FUNCTION_BLOCK CON_LoadingStation
VAR_INPUT
	i_weighbridge 					: MOD_Loadingstation_I_stWeighbridge;
	i_tempIWantExtraBoxInTruck 		: BOOL;
	i_resetTime						: TIME := T#2S;//time necessary for the slowest part to reset
END_VAR
VAR_OUTPUT
	q_crane 						: MOD_Loadingstation_Q_stCrane;
END_VAR
VAR_IN_OUT
	iq_CommandState 				: INT;
END_VAR
VAR
	resetTimer						: TON;
	resetState 						: INT;
END_VAR

//check if there is a truck before running. Also check for weightlimit
IF NOT i_weighbridge.TruckOnScale THEN
	q_crane.AllowedToOperate 	:= FALSE;
	iq_CommandState 			:= Command.Abort; //Abort no truck
	
ELSIF i_weighbridge.TruckOnScale AND NOT i_weighbridge.WeightLimitReached THEN
	q_crane.AllowedToOperate 	:= TRUE;//can come fromoutside?
	CASE resetState OF
		0:
			iq_CommandState 	:= Command.Reset;
			resetTimer(IN := TRUE, PT := i_resetTime);
			IF resetTimer.Q THEN
				resetTimer(IN := FALSE, PT := i_resetTime);
				resetState := 1;				
			END_IF
		1:
			iq_CommandState 	:= Command.Executing;
	END_CASE
// if operator wants an extra box loaded above the limit.
ELSIF i_tempIWantExtraBoxInTruck THEN //is supposed to be a button press
	q_crane.AllowedToOperate 	:= TRUE;
	CASE resetState OF
		0:
			iq_CommandState 	:= Command.Reset;
			resetTimer(IN := TRUE, PT := i_resetTime);
			IF resetTimer.Q THEN
				resetTimer(IN := FALSE, PT := i_resetTime);
				resetState := 1;				
			END_IF

		1:
			iq_CommandState 	:= Command.Executing;
	END_CASE
ELSIF i_weighbridge.WeightLimitReached THEN
	q_crane.AllowedToOperate 	:= FALSE;
	iq_CommandState 			:= Command.Stop;
	//done loading!
END_IF



CASE iq_CommandState OF
	Command.Abort:
		resetState := 0;
	Command.Reset:
		resetState := 0;
END_CASE

END_FUNCTION_BLOCK

(* stored: Version 1.1.0.1, ProductVersion 3.1.4024.6
   POU CON_LoadingStation: Id {fd02a03d-6b4a-42d7-8b82-6be1646338cc}, SpecialFunc None *)
